// TIA Portal V16 export
// export: Created 2021-11-15T21:16:57.6885547Z, ExportSetting WithDefaults, WithReadOnly, DisplayName Totally Integrated Automation Portal, DisplayVersion V16 Update 3, DisplayName TIA Portal Version Control Interface, DisplayVersion V16 Update 2, DisplayName TIA Portal Openness, DisplayVersion V16 Update 3, DisplayName SINAMICS Startdrive Advanced, DisplayVersion V16, DisplayName SINAMICS Startdrive G130, G150, S120, S150, SINAMICS MV, S210, DisplayVersion V16, DisplayName SINAMICS Startdrive G110M, G120, G120C, G120D, G120P, DisplayVersion V16, DisplayName STEP 7 Professional, DisplayVersion V16 Update 3, DisplayName SIMATIC Energy Suite, DisplayVersion V16, DisplayName STEP 7 Safety, DisplayVersion V16, DisplayName WinCC Advanced, DisplayVersion V16 Update 3
FUNCTION "Export" : Void   // FC2, LAD
{ S7_Optimized_Access := 'TRUE' }
VERSION : 0.1
// stored: AutoNumber true, CodeModifiedDate 2021-11-15T21:14:45.9278125Z, CompileDate 2021-11-15T21:14:56.9551563Z, CreationDate 2021-11-15T21:12:04.4639454Z, HandleErrorsWithinBlock false, InterfaceModifiedDate 2021-11-15T21:12:04.4639454Z, IsConsistent true, IsIECCheckEnabled false, IsKnowHowProtected false, IsWriteProtected false, LibraryConformanceStatus Avviso: Il blocco contiene accessi diretti a ingressi, uscite, merker, accessi indiretti a registri o accessi indiretti ad aree di memoria esterne sconosciute al momento della compilazione., ModifiedDate 2021-11-15T21:14:45.9278125Z, ParameterModified 2021-11-15T21:12:04.4639454Z, PLCSimAdvancedSupport true, SetENOAutomatically false, StructureModified 2021-11-15T21:12:04.4639454Z, UDAEnableTagReadback false
BEGIN

REGION Network 1
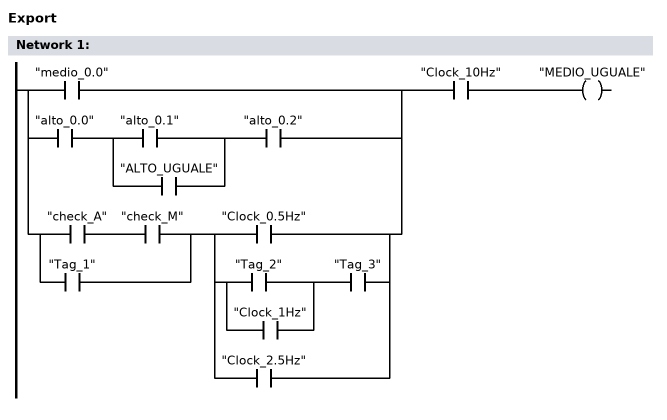
   RUNG wire#powerrail
      Contact( "medio_0.0" )
      wire#w1
      Contact( "Clock_10Hz" )
      Coil( "MEDIO_UGUALE" )
   END_RUNG
   RUNG wire#powerrail
      Contact( "alto_0.0" )
      wire#w2
      Contact( "alto_0.1" )
      wire#w3
      Contact( "alto_0.2" )
   END_RUNG wire#w1
   RUNG wire#w2
      Contact( "ALTO_UGUALE" )
   END_RUNG wire#w3
   RUNG wire#powerrail
      Contact( "check_A" )
      Contact( "check_M" )
      wire#w4
      Contact( "Clock_0.5Hz" )
   END_RUNG wire#w1
   RUNG wire#powerrail
      Contact( "Tag_1" )
   END_RUNG wire#w4
   RUNG wire#w4
      Contact( "Tag_2" )
      wire#w5
      Contact( "Tag_3" )
   END_RUNG wire#w1
   RUNG wire#w4
      Contact( "Clock_1Hz" )
   END_RUNG wire#w5
   RUNG wire#w4
      Contact( "Clock_2.5Hz" )
   END_RUNG wire#w1
   // the same network as SCL:
   "MEDIO_UGUALE" := ("medio_0.0" OR ("alto_0.0" AND ("alto_0.1" OR "ALTO_UGUALE") AND "alto_0.2") OR ((("check_A" AND "check_M") OR "Tag_1") AND ("Clock_0.5Hz" OR (("Tag_2" OR "Clock_1Hz") AND "Tag_3") OR "Clock_2.5Hz"))) AND "Clock_10Hz";
END_REGION
END_FUNCTION
